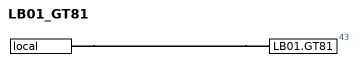
local := LB01.GT81;
ackFault S= local.ACK AND local.FAULT;
ackLal S= local.ACK AND local.LAL;
ackHal S= local.ACK AND local.HAL;
ackAl01 S= local.ACK AND local.AL01;
local.ACK R= true;
// Sensor error
AlarmAcknowledge01(
    Alarm := local.PV < -3200.0 AND NOT SYS_StartupDelayComm,
    InitPulse := SYS_InitPulse,
    AlarmAck := ackFault); // _BE_AlarmAckRemote
local.FAULT := AlarmAcknowledge01.AlarmActive;
// Alarm Low
gt_Min(IN := local.PV < local.ALL AND NOT SYS_StartupDelayComm AND LB01.GeneralStart AND NOT local.FAULT, PT := DINT_TO_TIME(local.AD * 60000)); // TON
AlarmAcknowledge02(Alarm := gt_Min.Q, InitPulse := SYS_InitPulse, AlarmAck := ackLal); // _BE_AlarmAckRemote
local.LAL := AlarmAcknowledge02.AlarmActive;
// Alarm High
gt_Max(IN := local.PV > local.AHL AND NOT SYS_StartupDelayComm AND LB01.GeneralStart AND NOT local.FAULT, PT := DINT_TO_TIME(local.AD * 60000)); // TON
AlarmAcknowledge03(Alarm := gt_Max.Q, InitPulse := SYS_InitPulse, AlarmAck := ackHal); // _BE_AlarmAckRemote
local.HAL := AlarmAcknowledge03.AlarmActive;
// Al01 - Freeze protection
AlarmFb01(Alarm := local.FreezeProtect AND NOT local.FAULT, InitPulse := SYS_InitPulse, AlarmAck := ackAl01); // _BE_AlarmAckRequired
local.AL01 := AlarmFb01.AlarmActive;
// General Alarm
local.AL := local.FAULT OR local.AL01;
// Status HMI
IF true THEN _w1 := 0; END_IF
local.Symbol := _w1;
IF local.FAULT OR local.LAL OR local.HAL OR local.FreezeProtect THEN _w2 := 2; END_IF
local.Symbol := _w2;
IF local.FAULT THEN _w3 := 3; END_IF
local.Symbol := _w3;
FbFreezeProt(
    Enable := NOT SYS_StartupDelayComm,
    SelectFunctionMode := LB01.GeneralStart,
    ProcessValueHeatingUnit := local.PV,
    SupportHeatingValue := local.SP2,
    FreezeProtectionValue := local.SP1,
    SetValueOffline := local.SP); // _BE_ReturnWaterControl
local.OP := FbFreezeProt.OutputValue;
local.FreezeProtect := FbFreezeProt.FreezeProtectionAlarm;
LB01.GT81 := local;

END_PROGRAM

// Device/AREA1/B001/LB01/Sensor/Temperature/GT31/LB01_GT31_Control
PROGRAM LB01_GT31_Control
VAR
	local:strSensor2_Regulator;
	gt_Min: TON;
	gt_Max: TON;
	reset_en: RS;
	FbRegulator: _BE_Regulator;
	ackFault: BOOL;
	ackLal: BOOL;
	ackHal: BOOL;
	AlarmAcknowledge01: _BE_AlarmAckRemote;
	AlarmAcknowledge02: _BE_AlarmAckRemote;
	AlarmAcknowledge03: _BE_AlarmAckRemote;
END_VAR
VAR // added by the converter: edge detectors and wires of the graphical bodies
    _w1, _w4, _w5, _w6, _w8, _w9 : ANY;
    _w2, _w3, _w7 : BOOL;
END_VAR

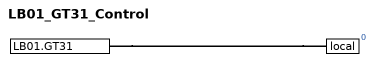
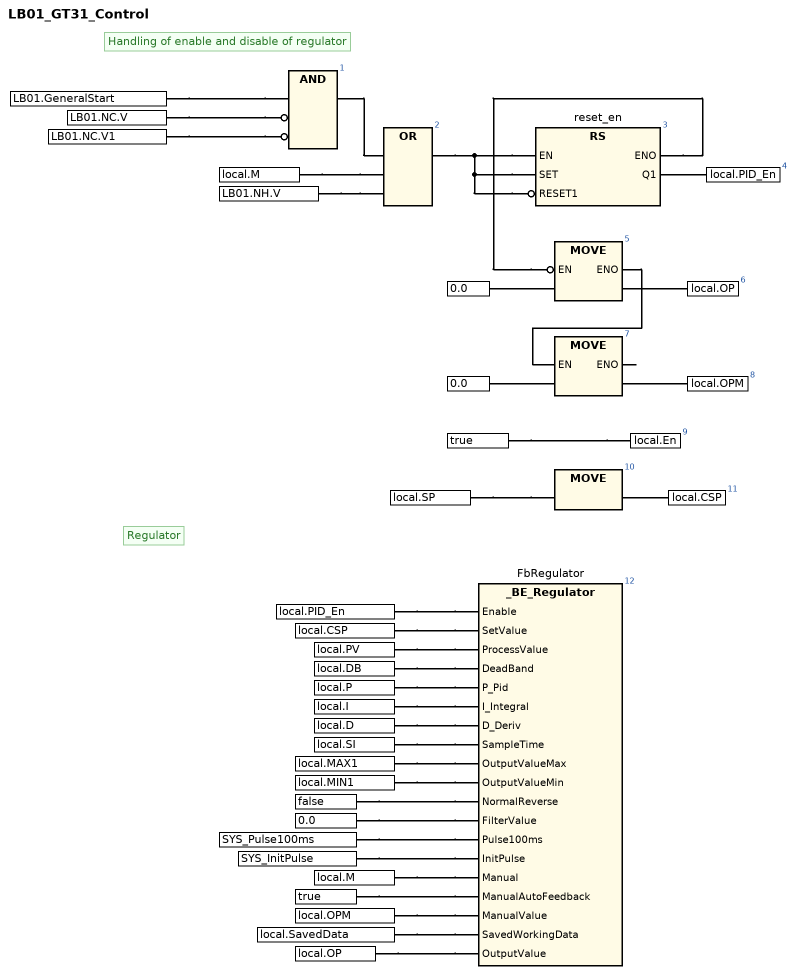
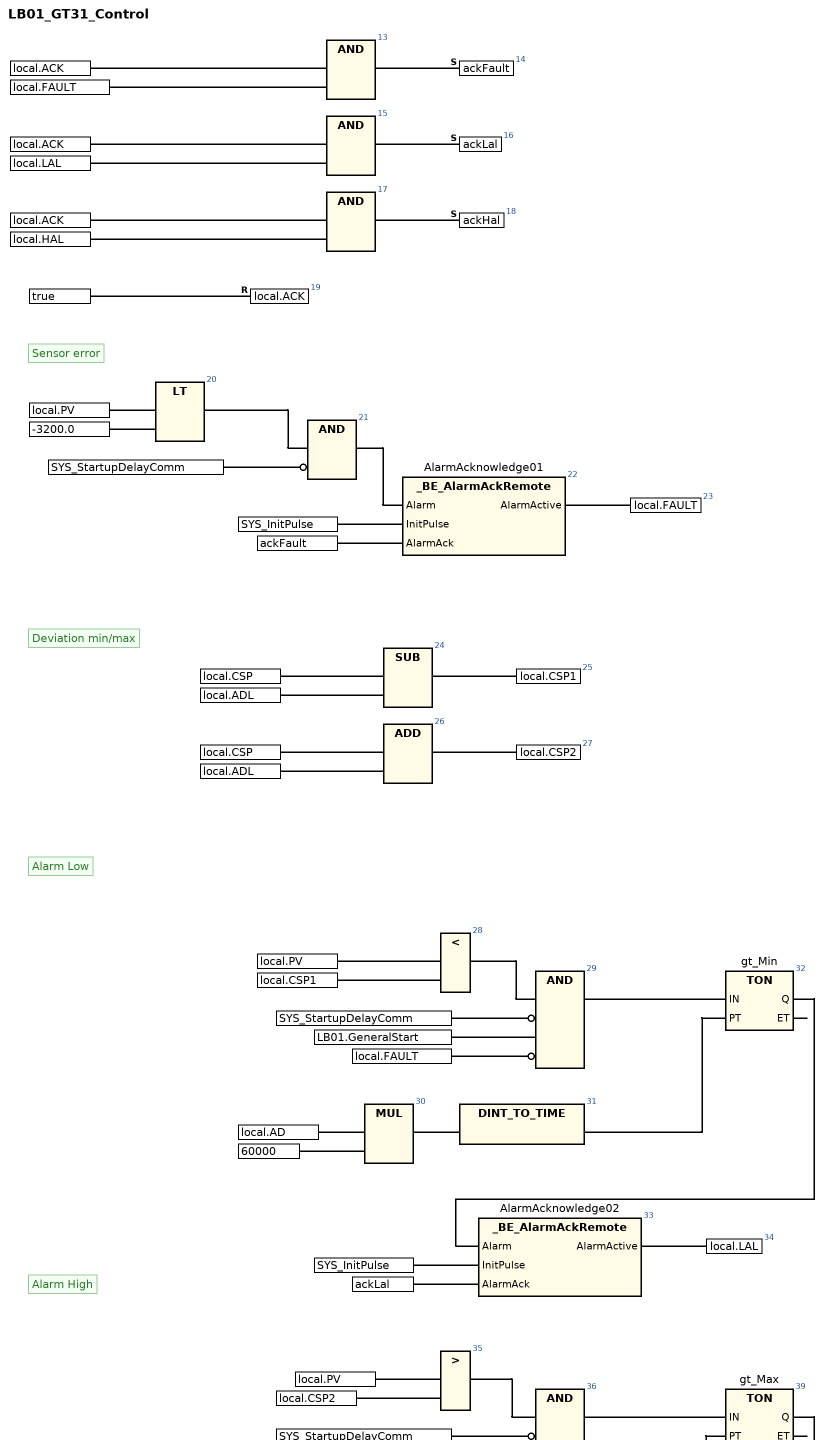
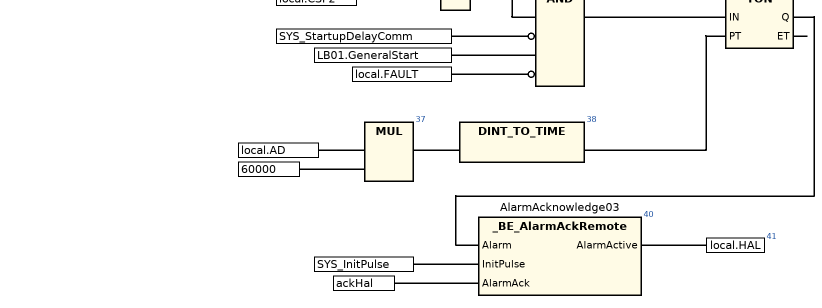
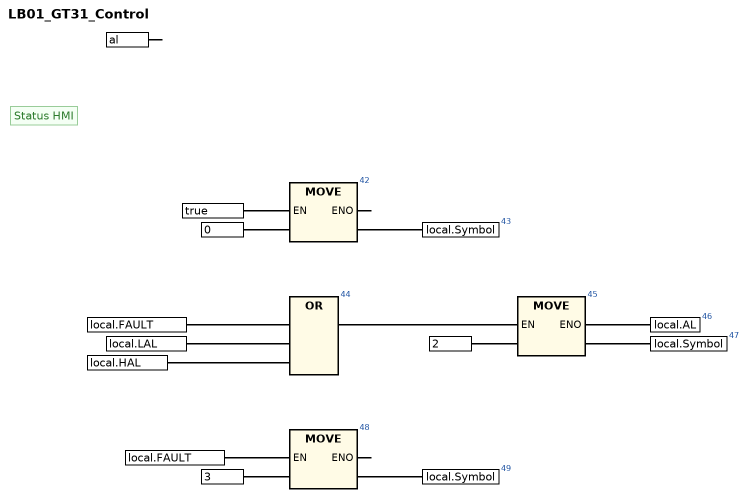
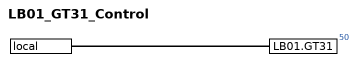
local := LB01.GT31;
// Handling of enable and disable of regulator
_w1 := LB01.GeneralStart AND NOT LB01.NC.V AND NOT LB01.NC.V1 OR local.M OR LB01.NH.V;
_w2 := _w1;
IF _w2 THEN
    reset_en(SET := _w1, RESET1 := NOT _w1); // RS
END_IF
local.PID_En := reset_en.Q1;
_w3 := NOT _w2;
IF _w3 THEN _w4 := 0.0; END_IF
local.OP := _w4;
IF _w3 THEN _w5 := 0.0; END_IF
local.OPM := _w5;
local.En := true;
local.CSP := local.SP;
// Regulator
FbRegulator(
    Enable := local.PID_En,
    SetValue := local.CSP,
    ProcessValue := local.PV,
    DeadBand := local.DB,
    P_Pid := local.P,
    I_Integral := local.I,
    D_Deriv := local.D,
    SampleTime := local.SI,
    OutputValueMax := local.MAX1,
    OutputValueMin := local.MIN1,
    NormalReverse := false,
    FilterValue := 0.0,
    Pulse100ms := SYS_Pulse100ms,
    InitPulse := SYS_InitPulse,
    Manual := local.M,
    ManualAutoFeedback := true,
    ManualValue := local.OPM,
    SavedWorkingData := local.SavedData,
    OutputValue := local.OP); // _BE_Regulator
ackFault S= local.ACK AND local.FAULT;
ackLal S= local.ACK AND local.LAL;
ackHal S= local.ACK AND local.HAL;
local.ACK R= true;
// Sensor error
AlarmAcknowledge01(
    Alarm := local.PV < -3200.0 AND NOT SYS_StartupDelayComm,
    InitPulse := SYS_InitPulse,
    AlarmAck := ackFault); // _BE_AlarmAckRemote
local.FAULT := AlarmAcknowledge01.AlarmActive;
// Deviation min/max
local.CSP1 := local.CSP - local.ADL;
local.CSP2 := local.CSP + local.ADL;
// Alarm Low
gt_Min(IN := local.PV < local.CSP1 AND NOT SYS_StartupDelayComm AND LB01.GeneralStart AND NOT local.FAULT, PT := DINT_TO_TIME(local.AD * 60000)); // TON
AlarmAcknowledge02(Alarm := gt_Min.Q, InitPulse := SYS_InitPulse, AlarmAck := ackLal); // _BE_AlarmAckRemote
local.LAL := AlarmAcknowledge02.AlarmActive;
// Alarm High
gt_Max(IN := local.PV > local.CSP2 AND NOT SYS_StartupDelayComm AND LB01.GeneralStart AND NOT local.FAULT, PT := DINT_TO_TIME(local.AD * 60000)); // TON
AlarmAcknowledge03(Alarm := gt_Max.Q, InitPulse := SYS_InitPulse, AlarmAck := ackHal); // _BE_AlarmAckRemote
local.HAL := AlarmAcknowledge03.AlarmActive;
// Status HMI
IF true THEN _w6 := 0; END_IF
local.Symbol := _w6;
_w7 := local.FAULT OR local.LAL OR local.HAL;
IF _w7 THEN _w8 := 2; END_IF
local.AL := _w7;
local.Symbol := _w8;
IF local.FAULT THEN _w9 := 3; END_IF
local.Symbol := _w9;
LB01.GT31 := local;
// al: input not connected

END_PROGRAM

// Device/AREA1/B001/LB01/Sensor/Temperature/GT31/LB01_Cascade_RoomControl
PROGRAM LB01_Cascade_RoomControl
VAR
END_VAR
VAR // added by the converter: edge detectors and wires of the graphical bodies
    _w1 : ANY;
END_VAR

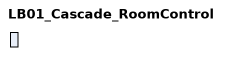
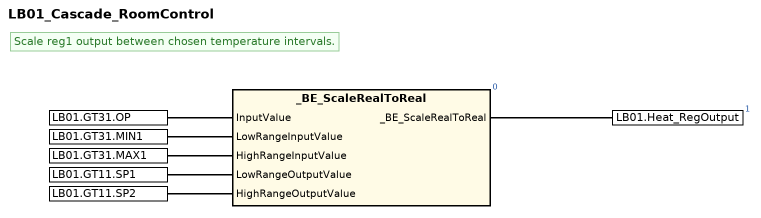
// Scale reg1 output between chosen temperature intervals.
_w1 := _BE_ScaleRealToReal(InputValue := LB01.GT31.OP, LowRangeInputValue := LB01.GT31.MIN1, HighRangeInputValue := LB01.GT31.MAX1, LowRangeOutputValue := LB01.GT11.SP1, HighRangeOutputValue := LB01.GT11.SP2);
LB01.Heat_RegOutput := _w1;

END_PROGRAM

// Device/AREA1/B001/LB01/Sensor/Temperature/GT11/LB01_GT11_RegHeating
PROGRAM LB01_GT11_RegHeating
VAR
	local:strSensor2_Regulator;
	gt_Min: TON;
	gt_Max: TON;
	reset_en: RS;
	FbRegulator: _BE_Regulator;
	cool_csp: REAL;
	cool_op: REAL;
	heatingOk: BOOL;
	sum_m: BOOL;
	tmp_opm: REAL;
END_VAR
VAR // added by the converter: edge detectors and wires of the graphical bodies
    _w1, _w2 : BOOL;
    _w3, _w4, _w5, _w6, _w7, _w8, _w9 : ANY;
END_VAR

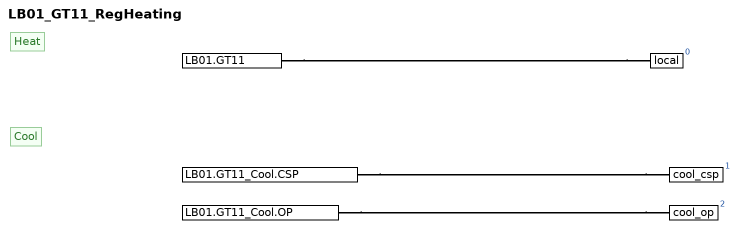
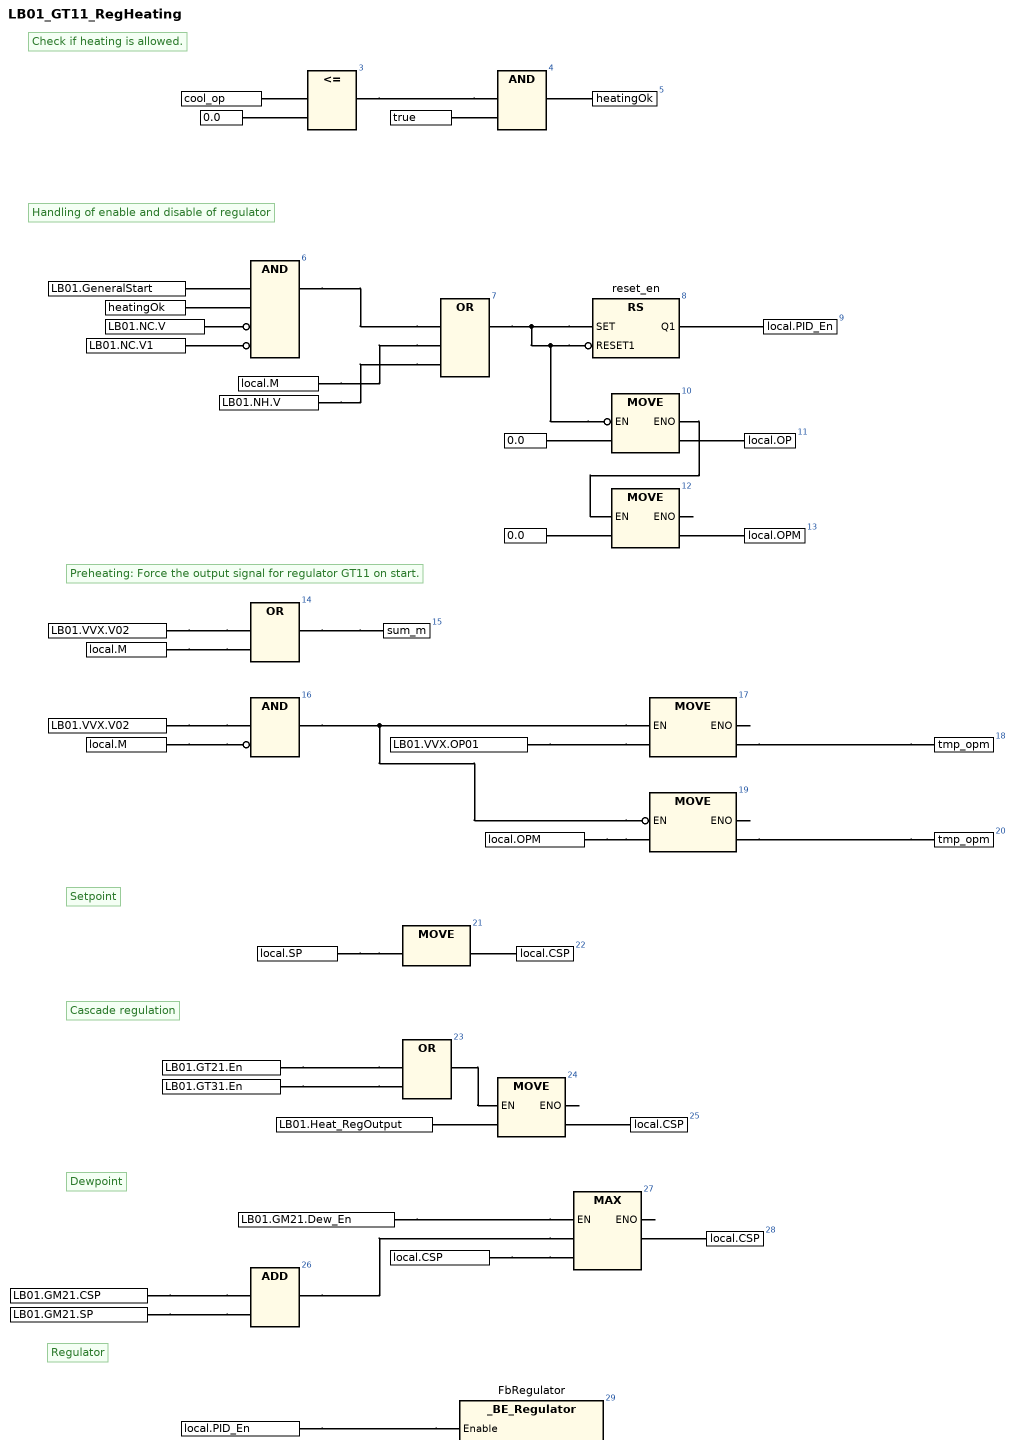
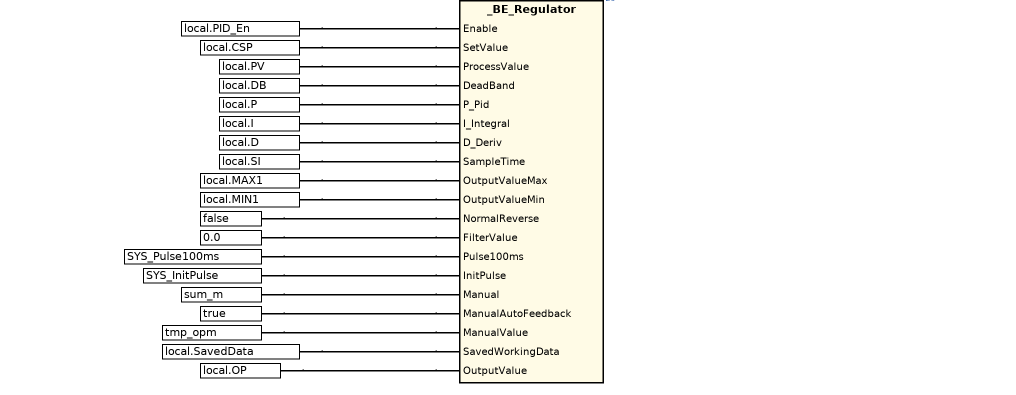
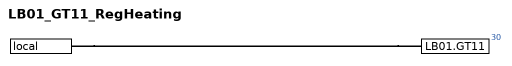
// Heat
local := LB01.GT11;
// Cool
cool_csp := LB01.GT11_Cool.CSP;
cool_op := LB01.GT11_Cool.OP;
// Check if heating is allowed.
heatingOk := cool_op <= 0.0 AND true;
// Handling of enable and disable of regulator
_w1 := LB01.GeneralStart AND heatingOk AND NOT LB01.NC.V AND NOT LB01.NC.V1 OR local.M OR LB01.NH.V;
reset_en(SET := _w1, RESET1 := NOT _w1); // RS
local.PID_En := reset_en.Q1;
_w2 := NOT _w1;
IF _w2 THEN _w3 := 0.0; END_IF
local.OP := _w3;
IF _w2 THEN _w4 := 0.0; END_IF
local.OPM := _w4;
// Preheating: Force the output signal for regulator GT11 on start.
sum_m := LB01.VVX.V02 OR local.M;
_w5 := LB01.VVX.V02 AND NOT local.M;
IF _w5 THEN _w6 := LB01.VVX.OP01; END_IF
tmp_opm := _w6;
IF NOT _w5 THEN _w7 := local.OPM; END_IF
tmp_opm := _w7;
// Setpoint
local.CSP := local.SP;
// Cascade regulation
IF LB01.GT21.En OR LB01.GT31.En THEN _w8 := LB01.Heat_RegOutput; END_IF
local.CSP := _w8;
// Dewpoint
IF LB01.GM21.Dew_En THEN _w9 := MAX(LB01.GM21.CSP + LB01.GM21.SP, local.CSP); END_IF
local.CSP := _w9;
// Regulator
FbRegulator(
    Enable := local.PID_En,
    SetValue := local.CSP,
    ProcessValue := local.PV,
    DeadBand := local.DB,
    P_Pid := local.P,
    I_Integral := local.I,
    D_Deriv := local.D,
    SampleTime := local.SI,
    OutputValueMax := local.MAX1,
    OutputValueMin := local.MIN1,
    NormalReverse := false,
    FilterValue := 0.0,
    Pulse100ms := SYS_Pulse100ms,
    InitPulse := SYS_InitPulse,
    Manual := sum_m,
    ManualAutoFeedback := true,
    ManualValue := tmp_opm,
    SavedWorkingData := local.SavedData,
    OutputValue := local.OP); // _BE_Regulator
LB01.GT11 := local;

END_PROGRAM

// Device/AREA1/B001/LB01/Sensor/Temperature/GT11/LB01_GT11_RegCooling
PROGRAM LB01_GT11_RegCooling
VAR
	local:strSensor2_Regulator;
	gt_Min: TON;
	gt_Max: TON;
	reset_en: RS;
	FbRegulator: _BE_Regulator;
	heat_csp: REAL;
	heat_op: REAL;
	coolingOk: BOOL;
	heat_pv: REAL;
END_VAR
VAR // added by the converter: edge detectors and wires of the graphical bodies
    _w1, _w2 : BOOL;
    _w3, _w4 : ANY;
    _w5 : REAL;
END_VAR

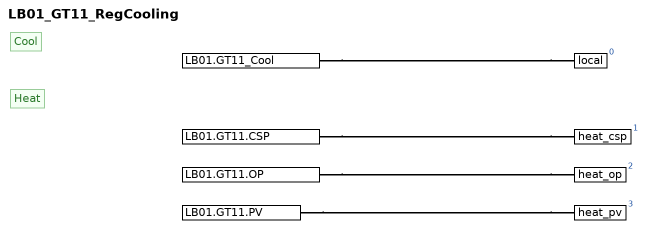
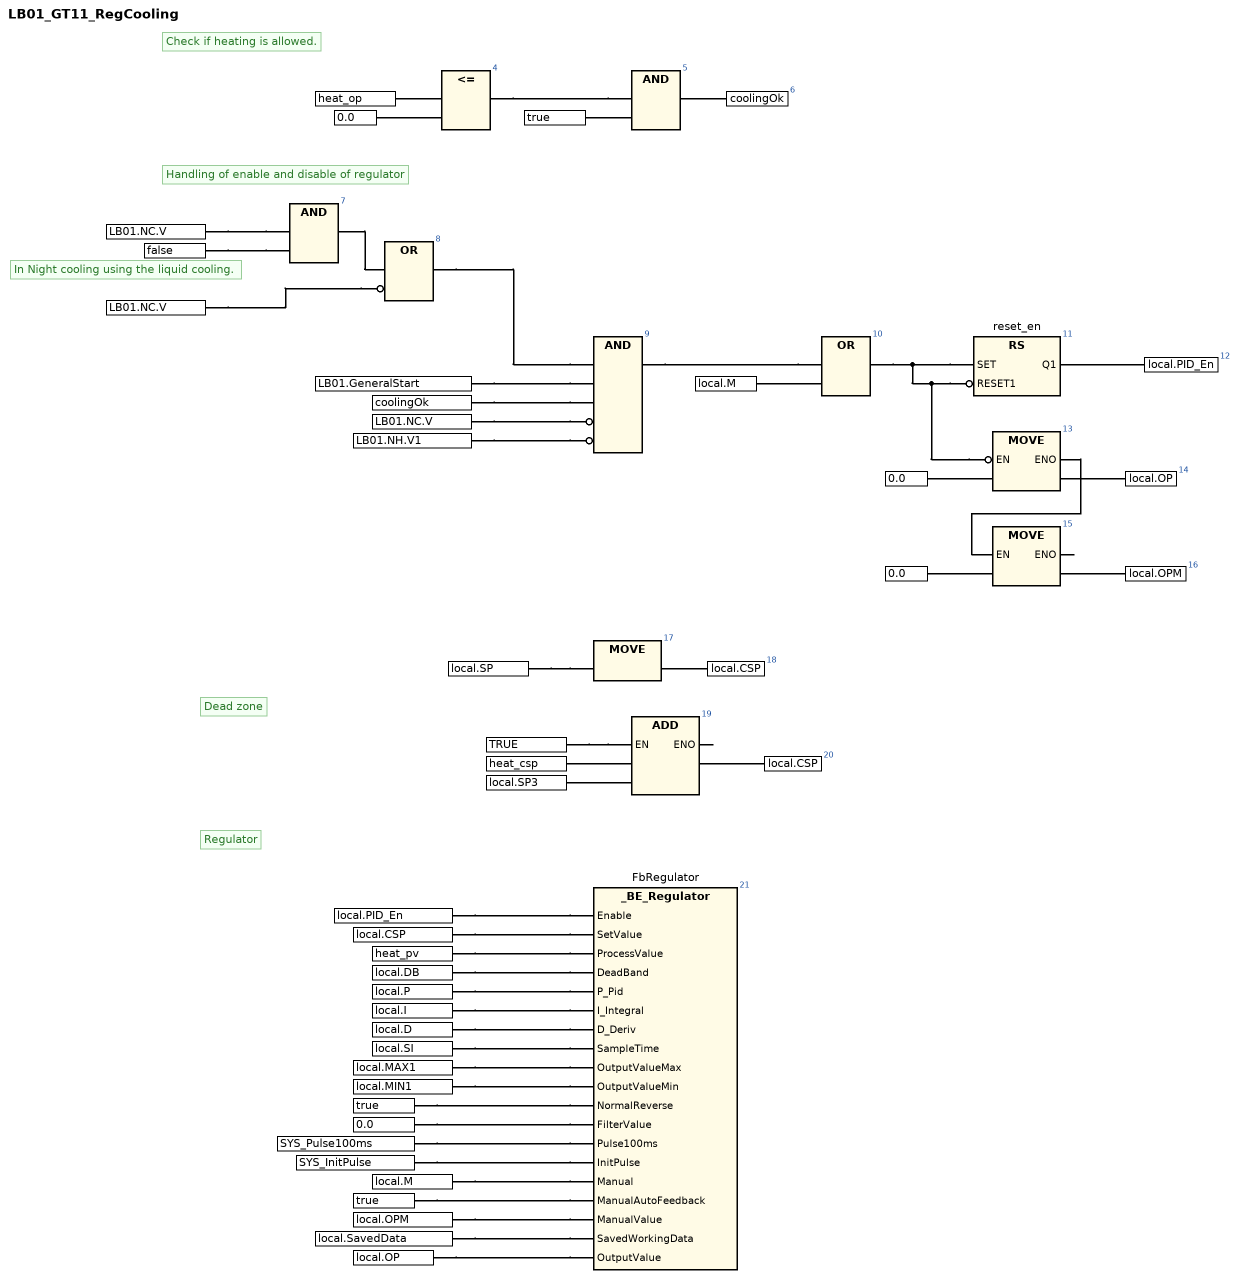
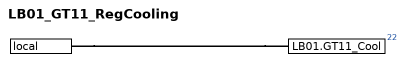
// Cool
local := LB01.GT11_Cool;
// Heat
heat_csp := LB01.GT11.CSP;
heat_op := LB01.GT11.OP;
heat_pv := LB01.GT11.PV;
// Check if heating is allowed.
coolingOk := heat_op <= 0.0 AND true;
// Handling of enable and disable of regulator
// In Night cooling using the liquid cooling.
_w1 := (LB01.NC.V AND false OR NOT LB01.NC.V) AND LB01.GeneralStart AND coolingOk AND NOT LB01.NC.V AND NOT LB01.NH.V1 OR local.M;
reset_en(SET := _w1, RESET1 := NOT _w1); // RS
local.PID_En := reset_en.Q1;
_w2 := NOT _w1;
IF _w2 THEN _w3 := 0.0; END_IF
local.OP := _w3;
IF _w2 THEN _w4 := 0.0; END_IF
local.OPM := _w4;
local.CSP := local.SP;
// Dead zone
_w5 := heat_csp + local.SP3;
local.CSP := _w5;
// Regulator
FbRegulator(
    Enable := local.PID_En,
    SetValue := local.CSP,
    ProcessValue := heat_pv,
    DeadBand := local.DB,
    P_Pid := local.P,
    I_Integral := local.I,
    D_Deriv := local.D,
    SampleTime := local.SI,
    OutputValueMax := local.MAX1,
    OutputValueMin := local.MIN1,
    NormalReverse := true,
    FilterValue := 0.0,
    Pulse100ms := SYS_Pulse100ms,
    InitPulse := SYS_InitPulse,
    Manual := local.M,
    ManualAutoFeedback := true,
    ManualValue := local.OPM,
    SavedWorkingData := local.SavedData,
    OutputValue := local.OP); // _BE_Regulator
LB01.GT11_Cool := local;

END_PROGRAM

// Device/AREA1/B001/LB01/Sensor/Temperature/GT11/LB01_GT11
PROGRAM LB01_GT11
VAR
	local:strSensor2_Regulator;
	gt_Min: TON;
	gt_Max: TON;
	reset_en: RS;
	ackFault: BOOL;
	ackLal: BOOL;
	ackHal: BOOL;
	AlarmAcknowledge01: _BE_AlarmAckRemote;
	AlarmAcknowledge02: _BE_AlarmAckRemote;
	AlarmAcknowledge03: _BE_AlarmAckRemote;
END_VAR
VAR // added by the converter: edge detectors and wires of the graphical bodies
    _w1, _w3, _w4 : ANY;
    _w2 : BOOL;
END_VAR

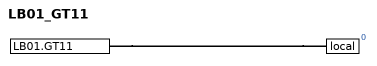
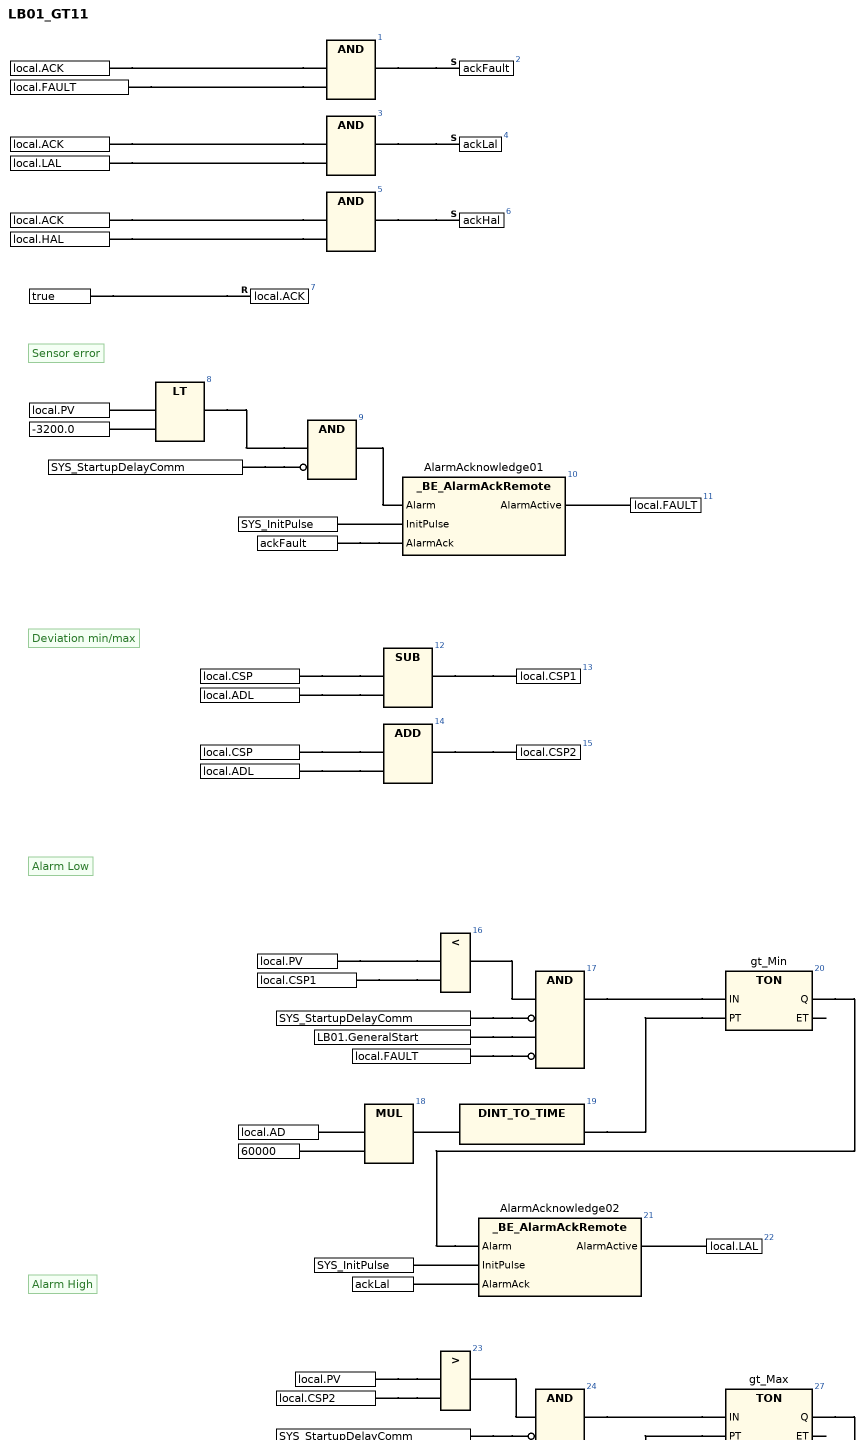
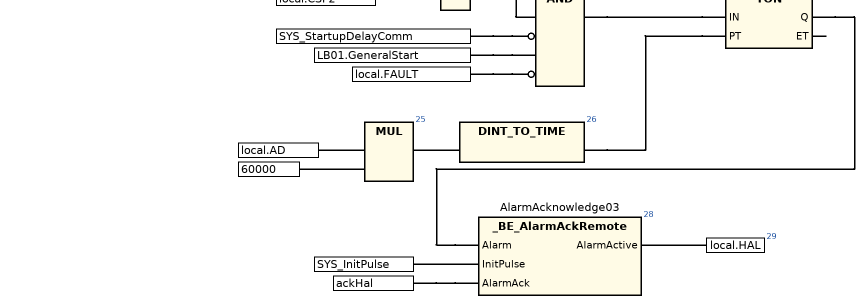
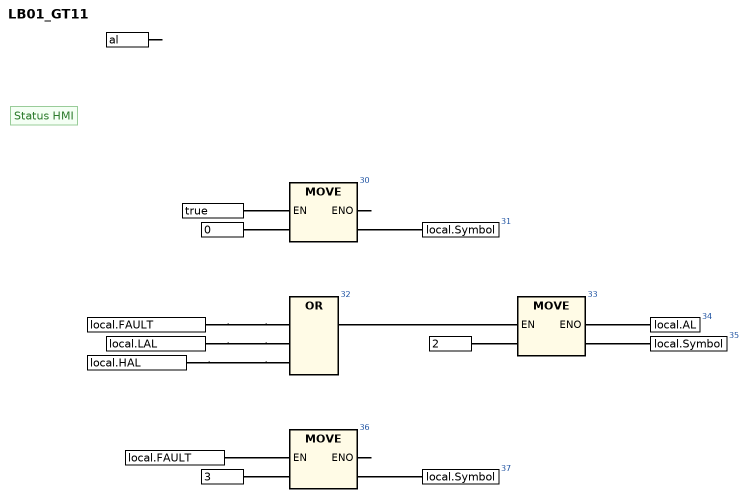
